FUNCTION INTERNAL _EmitSignal
VAR_INPUT
	iSignal		: I_SignalNode;
	iTag		: Tags.I_Tag;
END_VAR
VAR
	i			: UDINT;
	nEnd		: UDINT;
END_VAR

IF iSignal.count = 0 THEN
	RETURN;
END_IF

nEnd := iSignal.id + iSignal.count - 1;
FOR i := iSignal.id TO nEnd DO
	_Channel.stEntry[i].iReceiver.Receive(iTag);
END_FOR

END_FUNCTION

(* stored: Version 1.1.0.1
   POU _EmitSignal: Id {b87be85b-6104-4023-b85f-91882f5af811}, SpecialFunc None *)
